// TIA Portal project "练习1移动指令，转换指令_V16" (V16)

(* hardware
DEVICE "S7-1200 station_1"  S7-1200 Station
   slot 0: "Rack_0"  S7-1200 Rack  Rack  V1.0
   slot 1: "PLC_1"  CPU 1214C AC/DC/Rly  6ES7 214-1BG40-0XB0  V4.2
DEVICE "HMI_1"  KTP700 Basic PN
   slot 0: "HMI_1"  KTP700 Basic PN  6AV2 123-2GB03-0AX0  15.1.0.0
   slot 1: "HMI_RT_1"  KTP700 Basic PN  6AV2 123-2GB03-0AX0  15.1.0.0
   slot 5: "HMI_1.IE_CP_1"  PROFINET Interface  15.0.1.0
      slot 1: "PROFINET Interface_1"  PROFINET Interface
         slot 1: "Port_1"  Port
*)

// ===== PLC "PLC_1"  CPU 1214C AC/DC/Rly =====

VAR_GLOBAL   // PLC tag table "默认变量表"
   "Tag_1" AT %MD100 : UDInt;
   "Tag_2" AT %M0.0 : Bool;
   "Tag_3" AT %MD104 : UDInt;
   "Tag_4" AT %M0.1 : Bool;
END_VAR

DATA_BLOCK "日期"   // DB1
{ S7_Optimized_Access := 'TRUE' }
VERSION : 0.1
   VAR
      day_time : DTL;
      RET_VAL : Int;
      随机成绩 : UDInt;
      成绩 : Real;
      成绩1 : Real;
      成绩2 : UDInt;
      开关 : Bool;
      "数组1~10" : Array[1..10] of UDInt;
      转换数组2 : DInt;
      转换数组1 : DInt;
      开关1 : Bool;
      成绩3 : Real;
      总成绩 : UDInt;
      平均成绩变量 : Real;
      总成绩变量 : UDInt;
      开关2 : Bool;
      记录平均值的周期 : Bool;
      开关3 : Bool;
      初始化的周期 : Bool;
      录入成绩的周期 : Bool;
      "利用转换数组，将成绩数组归零" : UDInt;
      归零的平均成绩 : UDInt;
      带录入的成绩 : UDInt;
      录入成绩的标志 : UDInt;
   END_VAR
BEGIN
END_DATA_BLOCK

// folder: System blocks/Program resources

DATA_BLOCK "IEC_Counter_0_DB"   // DB2
{ S7_Optimized_Access := 'TRUE' }
AUTHOR : Simatic
FAMILY : IEC
NAME : CNTR
VERSION : 1.0
// stored: InstanceOfName IEC_COUNTER
"IEC_COUNTER"
BEGIN
END_DATA_BLOCK

// folder: (top level)

ORGANIZATION_BLOCK "Main"   // OB1, LAD, ProgramCycle
TITLE = "Main Program Sweep (Cycle)"
{ S7_Optimized_Access := 'TRUE' }
VERSION : 0.1
   VAR_INPUT
      Initial_Call : Bool;   // Initial call of this OB
      Remanence : Bool;   // =True, if remanent data are available
   END_VAR
   VAR_TEMP   // added for the SCL form of the ladder/FBD networks
      _w1 : Bool;
      _w2 : Bool;
      _w3 : Bool;
      _w4 : Bool;
   END_VAR
BEGIN

REGION Network 1: 随机生成一个成绩
   // 我们是利用日期这个数据块，选择其中的纳秒，为随机数,(利用时钟功能来确定)输出的日期
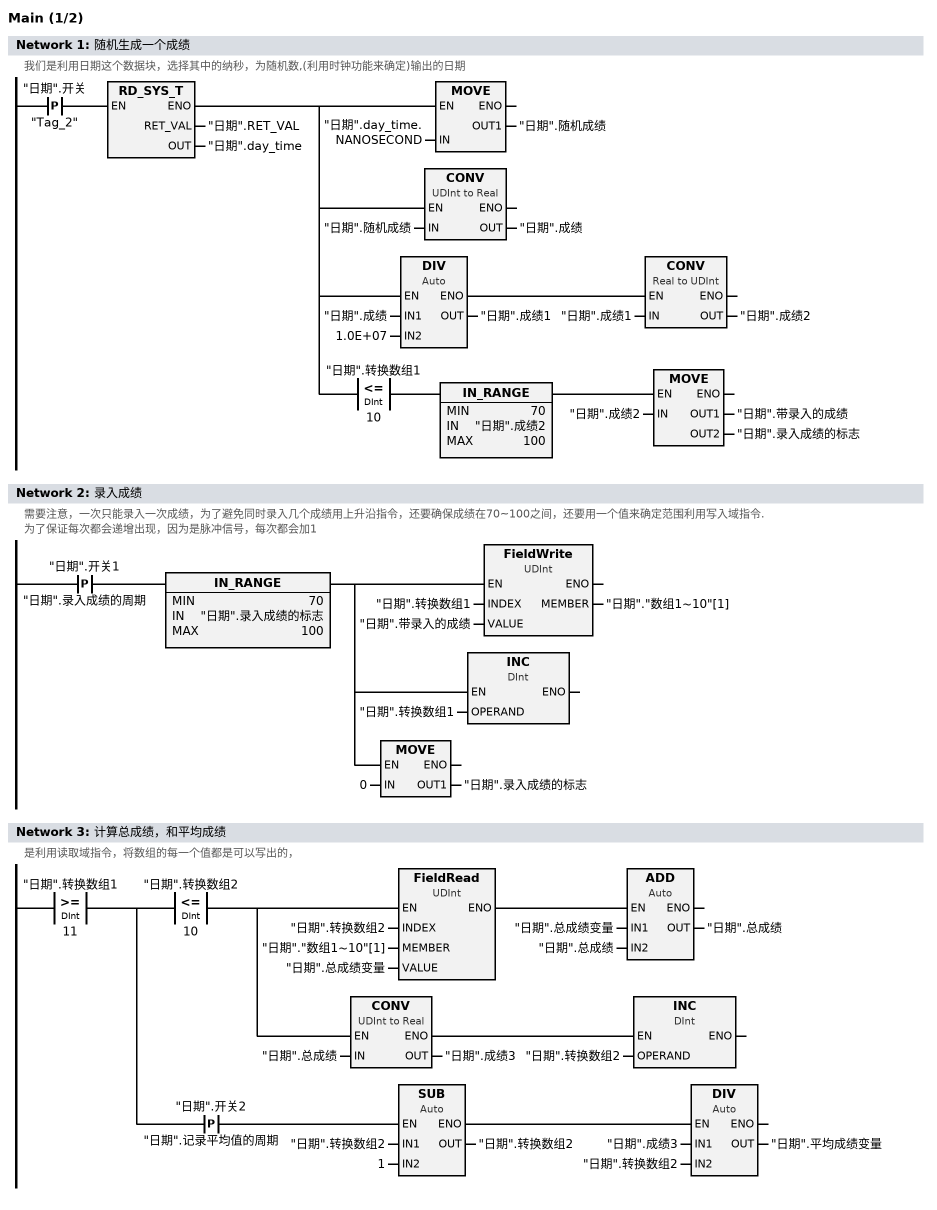
   // ENO of a box is taken as its EN; it also drops when the box reports an error
   #_w1 := "日期".开关 AND NOT "Tag_2";   // rising edge of "日期".开关
   "Tag_2" := "日期".开关;
   IF #_w1 THEN
       "日期".RET_VAL := RD_SYS_T(OUT => "日期".day_time);
       "日期".随机成绩 := "日期".day_time.NANOSECOND;
       "日期".成绩 := UDINT_TO_REAL("日期".随机成绩);
       "日期".成绩1 := "日期".成绩 / 1.0E+07;
       "日期".成绩2 := REAL_TO_UDINT("日期".成绩1);
   END_IF;
   IF #_w1 AND ("日期".转换数组1 <= 10) AND (70 <= "日期".成绩2) AND ("日期".成绩2 <= 100) THEN
       "日期".带录入的成绩 := "日期".成绩2;
       "日期".录入成绩的标志 := "日期".成绩2;
   END_IF;
END_REGION

REGION Network 2: 录入成绩
   // 需要注意，一次只能录入一次成绩，为了避免同时录入几个成绩用上升沿指令，还要确保成绩在70~100之间，还要用一个值来确定范围利用写入域指令.为了保证每次都会递增出现，因为是脉冲信号，每次都会加1
   // no SCL statement known for FieldWrite: written as a call
   #_w1 := "日期".开关1 AND NOT "日期".录入成绩的周期;   // rising edge of "日期".开关1
   "日期".录入成绩的周期 := "日期".开关1;
   #_w2 := #_w1 AND (70 <= "日期".录入成绩的标志) AND ("日期".录入成绩的标志 <= 100);
   IF #_w2 THEN
       FieldWrite(index := "日期".转换数组1, value := "日期".带录入的成绩, member => "日期"."数组1~10"[1]);
       "日期".转换数组1 := "日期".转换数组1 + 1;
       "日期".录入成绩的标志 := 0;
   END_IF;
END_REGION

REGION Network 3: 计算总成绩，和平均成绩
   // 是利用读取域指令，将数组的每一个值都是可以写出的，
   // no SCL statement known for FieldRead: written as a call
   // ENO of a box is taken as its EN; it also drops when the box reports an error
   #_w1 := "日期".转换数组1 >= 11;
   #_w2 := #_w1 AND ("日期".转换数组2 <= 10);
   #_w3 := #_w1 AND ("日期".转换数组2 <= 10);
   IF #_w3 THEN
       FieldRead(index := "日期".转换数组2, member := "日期"."数组1~10"[1], value := "日期".总成绩变量);
       "日期".总成绩 := "日期".总成绩变量 + "日期".总成绩;
   END_IF;
   IF #_w2 THEN
       "日期".成绩3 := UDINT_TO_REAL("日期".总成绩);
       "日期".转换数组2 := "日期".转换数组2 + 1;
   END_IF;
   #_w4 := #_w1 AND "日期".开关2 AND NOT "日期".记录平均值的周期;   // rising edge of "日期".开关2
   "日期".记录平均值的周期 := "日期".开关2;
   IF #_w4 THEN
       "日期".转换数组2 := "日期".转换数组2 - 1;
       "日期".平均成绩变量 := "日期".成绩3 / "日期".转换数组2;
   END_IF;
END_REGION

REGION Network 4: 初始化成绩
   // 要将，逐渐增加的变量，改变成绩的转换数组清零，要将数组里面的成绩全部清零，主要还要将之前，在计算成绩之间的转换数据类型的也要归零
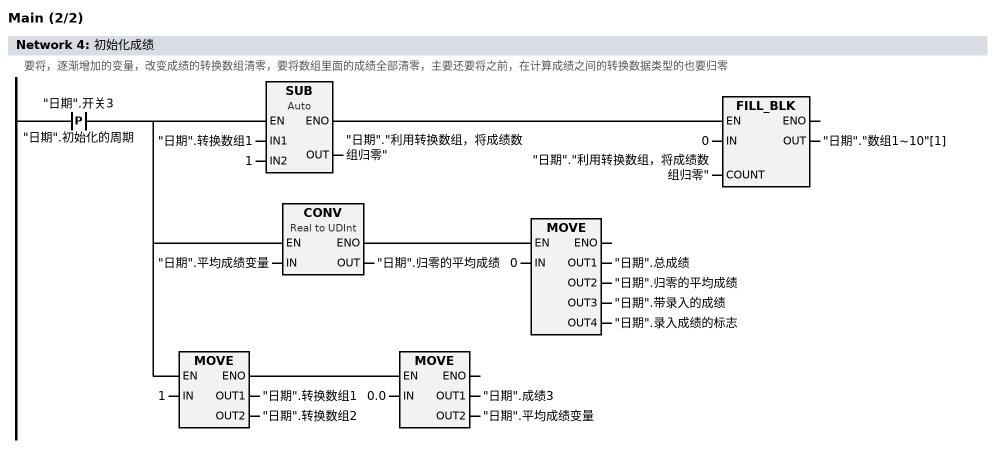
   RUNG wire#powerrail
      P_Contact(operand := "日期".开关3, bit := "日期".初始化的周期)
      wire#w1
      Sub(in1 := "日期".转换数组1, in2 := 1, out => "日期"."利用转换数组，将成绩数组归零")
      FillBlockI(in := 0, count := "日期"."利用转换数组，将成绩数组归零", out => "日期"."数组1~10"[1])
   END_RUNG
   RUNG wire#w1
      { S7_Templates := "[SrcType := Real, DestType := UDInt]" } Convert(in := "日期".平均成绩变量, out => "日期".归零的平均成绩)
      Move(in := 0, out1 => "日期".总成绩, out2 => "日期".归零的平均成绩, out3 => "日期".带录入的成绩, out4 => "日期".录入成绩的标志)
   END_RUNG
   RUNG wire#w1
      Move(in := 1, out1 => "日期".转换数组1, out2 => "日期".转换数组2)
      Move(in := 0.0, out1 => "日期".成绩3, out2 => "日期".平均成绩变量)
   END_RUNG
   // the same network as SCL:
   #_w1 := "日期".开关3 AND NOT "日期".初始化的周期;   // rising edge of "日期".开关3
   "日期".初始化的周期 := "日期".开关3;
   IF #_w1 THEN
       "日期"."利用转换数组，将成绩数组归零" := "日期".转换数组1 - 1;
       FILL_BLK(IN := 0, COUNT := "日期"."利用转换数组，将成绩数组归零", OUT => "日期"."数组1~10"[1]);
       "日期".归零的平均成绩 := REAL_TO_UDINT("日期".平均成绩变量);
       "日期".总成绩 := 0;
       "日期".归零的平均成绩 := 0;
       "日期".带录入的成绩 := 0;
       "日期".录入成绩的标志 := 0;
       "日期".转换数组1 := 1;
       "日期".转换数组2 := 1;
       "日期".成绩3 := 0.0;
       "日期".平均成绩变量 := 0.0;
   END_IF;
END_REGION
END_ORGANIZATION_BLOCK

(* ===== HMI "HMI_RT_1" =====
system functions are stored by id; their names below are inferred from use
connection "HMI_连接_1": ETHERNET, SMART_S7_1200_OMS
connection "HMI_连接_2": ETHERNET, SMART_S7_1200_OMS

HMI tags "默认变量表"
   "Tag_ScreenNumber" : UInt, internal
   "日期_开关" : Bool = PLC 日期.开关, 1 s
   "日期_开关1" : Bool = PLC 日期.开关1, 1 s
   "日期_开关2" : Bool = PLC 日期.开关2, 1 s
   "日期_开关3" : Bool = PLC 日期.开关3, 1 s
   "Tag_1" : UDInt = PLC Tag_1 AT %MD100, 1 s
   "日期_平均成绩变量" : Real = PLC 日期.平均成绩变量, 1 s
   "日期_带录入的成绩" : UDInt = PLC 日期.带录入的成绩, 1 s
   "日期_转换数组1" : DInt = PLC 日期.转换数组1, 1 s

Template "模板_1" 800x480
   Button "退出" at 714,429 size 71x50; TextOff '退出'; PictureOff "ExitRuntime_KTP700_Basic_PN_TR"; PictureOn "ExitRuntime_KTP700_Basic_PN_TR"
      on Release: StopRuntime(0)
   Button "Template_Button" at 614,429 size 71x50; TextOff 'Text'
   Button "Template_Button_1" at 514,429 size 71x50; TextOff 'Text'
   Button "Template_Button_2" at 414,429 size 71x50; TextOff 'Text'
   Button "Template_Button_3" at 314,429 size 71x50; TextOff 'Text'
   Button "Template_Button_4" at 214,429 size 71x50; TextOff 'Text'
   Button "Template_Button_5" at 114,429 size 71x50; TextOff 'Text'
   Button "起始画面" at 14,429 size 71x50; TextOff '起始画面'; PictureOff "NavigateHome_KTP700_Basic_PN_TR"; PictureOn "NavigateHome_KTP700_Basic_PN_TR"
      on Release: ActivateScreen("根画面", 0)
   SymbolicIOField "Symbolic_IO_Field_Screen" at 93,9 size 600x33; TextOff '0'; TextOn '1'; TextList "TextList_ScreenNames"
      ProcessValue <- "Tag_ScreenNumber"
      on Change: ActivateScreenByNumber("Tag_ScreenNumber", 0)
   DateTimeField "HmiScreenItemData" at 695,25 size 105x25
   DateTimeField "HmiScreenItemData_1" at 695,0 size 105x25
   GraphicView "Logo" at 0,0 size 91x51; Picture "HMI_1 的 Logo"

screen "根画面" 800x480, template "模板_1"
   on GenerateScreen: SetTag("Tag_ScreenNumber", 1)
   TextField "文本域_1" at 258,63 size 307x33; Text '计算10同学的平均成绩'
      Visibility <- "日期_转换数组1"
   Button "按钮_1" at 146,270 size 133x55; TextOff '生成成绩'
      on Press: SetBit("日期_开关")
      on Release: ResetBit("日期_开关")
   Button "按钮_2" at 146,359 size 133x55; TextOff '录入成绩'
      on Release: ResetBit("日期_开关1")
      on Press: SetBit("日期_开关1")
   Button "按钮_3" at 455,270 size 133x55; TextOff '平均成绩'
      on Press: SetBit("日期_开关2")
      on Release: ResetBit("日期_开关2")
   Button "按钮_4" at 456,359 size 133x55; TextOff '初始化'
      on Release: ResetBit("日期_开关3")
      on Press: SetBit("日期_开关3")
   IOField "I/O 域_1" at 151,156 size 128x57; FormatPattern 99
      ProcessValue <- "日期_带录入的成绩"
   IOField "I/O 域_2" at 470,156 size 128x57; FormatPattern s99.9
      ProcessValue <- "日期_平均成绩变量"
*)